// TIA Portal V16 export
// export: Created 2020-03-06T18:52:04.504784Z, ExportSetting WithDefaults, DisplayName Totally Integrated Automation Portal, DisplayVersion V16, DisplayName TIA Portal Version Control Interface, DisplayVersion V16, DisplayName TIA Portal Openness, DisplayVersion V16, DisplayName TIA Portal Teamcenter Gateway, DisplayVersion V16, DisplayName SINAMICS Startdrive Advanced, DisplayVersion V16 Update 1, DisplayName SINAMICS Startdrive G130, G150, S120, S150, SINAMICS MV, S210, DisplayVersion V16 Update 1, DisplayName SINAMICS Startdrive G110M, G120, G120C, G120D, G120P, DisplayVersion V16 Update 1, DisplayName STEP 7 Professional, DisplayVersion V16, DisplayName STEP 7 Safety, DisplayVersion V16, DisplayName WinCC Professional, DisplayVersion V16
FUNCTION_BLOCK "3oo6 AI"   // FB37, LAD
{ S7_Optimized_Access := 'TRUE' }
VERSION : 0.1
// stored: AutoNumber true, IsIECCheckEnabled false, IsRetainMemResEnabled false, MemoryReserve 100, SetENOAutomatically false, UDAEnableTagReadback false
   VAR_INPUT
      V1GA : Bool;   // Value 1
      V2GA : Bool;   // Value 2
      V3GA : Bool;   // Value 3
      V4GA : Bool;
      V5GA : Bool;
      V6GA : Bool;
      "AL.HH3oo6" : Bool;
      "AL.H3oo6" : Bool;
      "AL.L3oo6" : Bool;
      "AL.LL3oo6" : Bool;
      PM : Int;   // Permissive Mode - "0=No P""1=Bool P" "2=Real P"
      HPB : Bool := TRUE;   // High Permissive BOOL
      LPB : Bool := TRUE;   // Low Permissive BOOL
      HPR : Real;   // High Permissive REAL
      LPR : Real;   // Low Permissive REAL
   END_VAR
   VAR_OUTPUT
      V1GA_1 : Bool;   // Value 1
      V2GA_1 : Bool;   // Value 2
      V3GA_1 : Bool;   // Value 3
      V4GA_1 : Bool;
      V5GA_1 : Bool;
      V6GA_1 : Bool;
      "AL.HH_3oo6" : Bool;
      "AL.H_3oo6" : Bool;
      "AL.L_3oo6" : Bool;
      "AL.LL_3oo6" : Bool;
   END_VAR
   VAR DB_SPECIFIC
      Config : Struct   // Configurations
         Limits : Struct
            HH : Real := 100.0;   // High High Limit
            H : Real := 90.0;   // High Limit
            L : Real := 10.0;   // Low Limit
            LL : Real := 5.0;   // Low Low Limit
         END_STRUCT;
         H : Real := 1.0;   // Hysteresis
      END_STRUCT;
      Alarms : Struct
         HH : Bool;   // High High
         H : Bool;   // High
         L : Bool;   // Low
         LL : Bool;   // Low Low
         V1GA : Bool;   // Value 1 General Alarm
         V2GA : Bool;   // Value 2 General Alarm
         V3GA : Bool;   // Value 3 General Alarm
         V4GA : Bool;
         V5GA : Bool;
         V6GA : Bool;
      END_STRUCT;
   END_VAR
   VAR
      V1HHA { ExternalAccessible := 'False'; ExternalVisible := 'False'; ExternalWritable := 'False'} : "HLR";   // Value 1 High High Alarm
      V1HA { ExternalAccessible := 'False'; ExternalVisible := 'False'; ExternalWritable := 'False'} : "HLR";   // Value 1 High Alarm
      V1LA { ExternalAccessible := 'False'; ExternalVisible := 'False'; ExternalWritable := 'False'} : "LLR";   // Value 1 Low Alarm
      V1LLA { ExternalAccessible := 'False'; ExternalVisible := 'False'; ExternalWritable := 'False'} : "LLR";   // Value 1 Low Low Alarm
      V2HHA { ExternalAccessible := 'False'; ExternalVisible := 'False'; ExternalWritable := 'False'} : "HLR";   // Value 2 High High Alarm
      V2HA { ExternalAccessible := 'False'; ExternalVisible := 'False'; ExternalWritable := 'False'} : "HLR";   // Value 2 High Alarm
      V2LA { ExternalAccessible := 'False'; ExternalVisible := 'False'; ExternalWritable := 'False'} : "LLR";   // Value 2 Low Alarm
      V2LLA { ExternalAccessible := 'False'; ExternalVisible := 'False'; ExternalWritable := 'False'} : "LLR";   // Value 2 Low Low Alarm
      V3HHA { ExternalAccessible := 'False'; ExternalVisible := 'False'; ExternalWritable := 'False'} : "HLR";   // Value 3 High High Alarm
      V3HA { ExternalAccessible := 'False'; ExternalVisible := 'False'; ExternalWritable := 'False'} : "HLR";   // Value 3 High Alarm
      V3LA { ExternalAccessible := 'False'; ExternalVisible := 'False'; ExternalWritable := 'False'} : "LLR";   // Value 3 Low Alarm
      V3LLA { ExternalAccessible := 'False'; ExternalVisible := 'False'; ExternalWritable := 'False'} : "LLR";   // Value 3 Low Low Alarm
   END_VAR
   VAR DB_SPECIFIC
      "HMI.FVR" : Real := 100.0;
      "FVR.HH" : DInt;
      "FVR.H" : DInt;
      "FVR.L" : DInt;
      "FVR.LL" : DInt;
      "FVR.HPR" : DInt;
      "FVR.LPR" : DInt;
      "FVR.CONFIG.H" : DInt;
   END_VAR
   VAR
      V4HHA { ExternalAccessible := 'False'; ExternalVisible := 'False'; ExternalWritable := 'False'} : "HLR";
      V4HA { ExternalAccessible := 'False'; ExternalVisible := 'False'; ExternalWritable := 'False'} : "HLR";
      V4LA { ExternalAccessible := 'False'; ExternalVisible := 'False'; ExternalWritable := 'False'} : "LLR";
      V4LLA { ExternalAccessible := 'False'; ExternalVisible := 'False'; ExternalWritable := 'False'} : "LLR";
      V6LLA { ExternalAccessible := 'False'; ExternalVisible := 'False'; ExternalWritable := 'False'} : "LLR";
      V6LA { ExternalAccessible := 'False'; ExternalVisible := 'False'; ExternalWritable := 'False'} : "LLR";
      V6HA { ExternalAccessible := 'False'; ExternalVisible := 'False'; ExternalWritable := 'False'} : "HLR";
      V6HHA { ExternalAccessible := 'False'; ExternalVisible := 'False'; ExternalWritable := 'False'} : "HLR";
      V5LLA { ExternalAccessible := 'False'; ExternalVisible := 'False'; ExternalWritable := 'False'} : "LLR";
      V5LA { ExternalAccessible := 'False'; ExternalVisible := 'False'; ExternalWritable := 'False'} : "LLR";
      V5HA { ExternalAccessible := 'False'; ExternalVisible := 'False'; ExternalWritable := 'False'} : "HLR";
      V5HHA { ExternalAccessible := 'False'; ExternalVisible := 'False'; ExternalWritable := 'False'} : "HLR";
   END_VAR
   VAR_TEMP
      HH123 : Bool;
      HH124 : Bool;
      HH134 : Bool;
      HH234 : Bool;
      HH125 : Bool;
      HH135 : Bool;
      HH235 : Bool;
      HH145 : Bool;
      HH245 : Bool;
      HH345 : Bool;
      HH126 : Bool;
      HH136 : Bool;
      HH236 : Bool;
      HH146 : Bool;
      HH246 : Bool;
      HH346 : Bool;
      HH156 : Bool;
      HH256 : Bool;
      HH356 : Bool;
      HH456 : Bool;
      H123 : Bool;
      H124 : Bool;
      H134 : Bool;
      H234 : Bool;
      H125 : Bool;
      H135 : Bool;
      H235 : Bool;
      H145 : Bool;
      H245 : Bool;
      H345 : Bool;
      H126 : Bool;
      H136 : Bool;
      H236 : Bool;
      H146 : Bool;
      H246 : Bool;
      H346 : Bool;
      H156 : Bool;
      H256 : Bool;
      H356 : Bool;
      H456 : Bool;
      L123 : Bool;
      L124 : Bool;
      L134 : Bool;
      L234 : Bool;
      L125 : Bool;
      L135 : Bool;
      L235 : Bool;
      L145 : Bool;
      L245 : Bool;
      L345 : Bool;
      L126 : Bool;
      L136 : Bool;
      L236 : Bool;
      L146 : Bool;
      L246 : Bool;
      L346 : Bool;
      L156 : Bool;
      L256 : Bool;
      L356 : Bool;
      L456 : Bool;
      LL123 : Bool;
      LL124 : Bool;
      LL134 : Bool;
      LL234 : Bool;
      LL125 : Bool;
      LL135 : Bool;
      LL235 : Bool;
      LL145 : Bool;
      LL245 : Bool;
      LL345 : Bool;
      LL126 : Bool;
      LL136 : Bool;
      LL236 : Bool;
      LL146 : Bool;
      LL246 : Bool;
      LL346 : Bool;
      LL156 : Bool;
      LL256 : Bool;
      LL356 : Bool;
      LL456 : Bool;
      "MATH.HH" : Real;
      "MATH.H" : Real;
      "MATH.LL" : Real;
      "MATH.L" : Real;
      "MATH.HR" : Real;
      "MATH.LR" : Real;
      "MATH.CONFIG.H" : Real;
   END_VAR
BEGIN

REGION Network 1
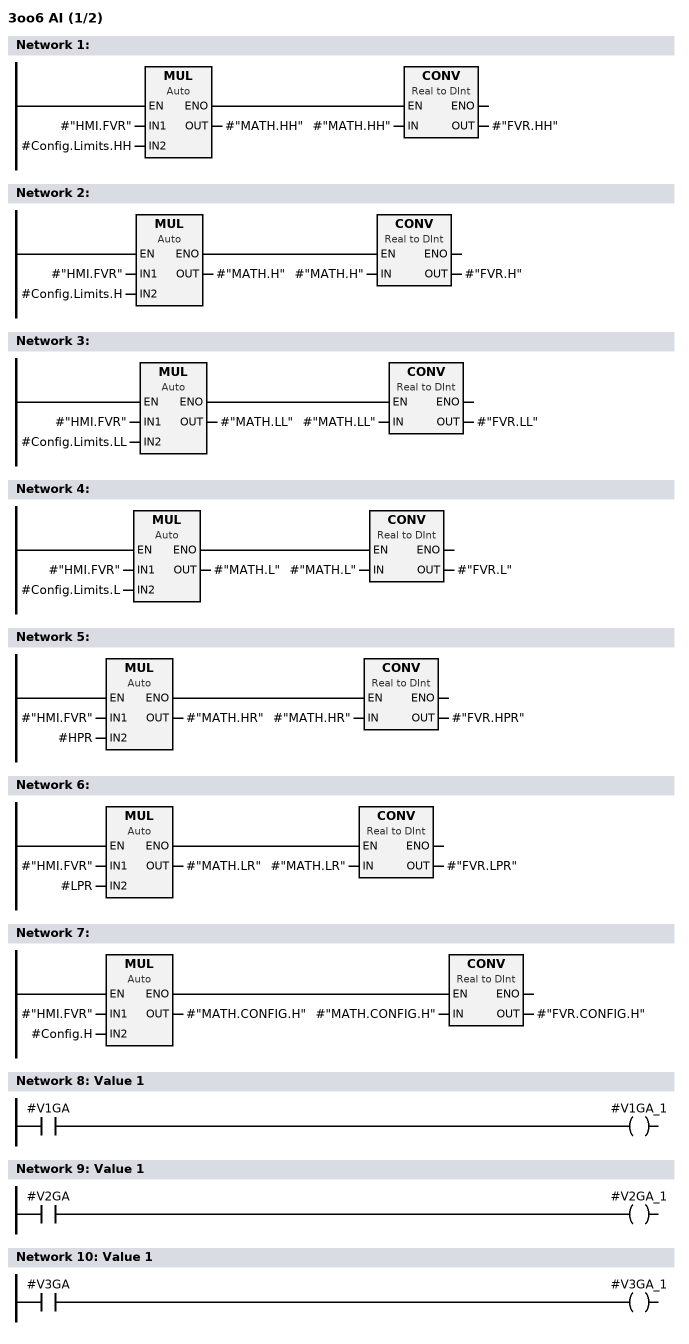
   RUNG wire#powerrail
      Mul(in1 := #"HMI.FVR", in2 := #Config.Limits.HH, out => #"MATH.HH")
      { S7_Templates := "[SrcType := Real, DestType := DInt]" } Convert(in := #"MATH.HH", out => #"FVR.HH")
   END_RUNG
   // the same network as SCL:
   #"MATH.HH" := #"HMI.FVR" * #Config.Limits.HH;
   #"FVR.HH" := REAL_TO_DINT(#"MATH.HH");
END_REGION

REGION Network 2
   RUNG wire#powerrail
      Mul(in1 := #"HMI.FVR", in2 := #Config.Limits.H, out => #"MATH.H")
      { S7_Templates := "[SrcType := Real, DestType := DInt]" } Convert(in := #"MATH.H", out => #"FVR.H")
   END_RUNG
   // the same network as SCL:
   #"MATH.H" := #"HMI.FVR" * #Config.Limits.H;
   #"FVR.H" := REAL_TO_DINT(#"MATH.H");
END_REGION

REGION Network 3
   RUNG wire#powerrail
      Mul(in1 := #"HMI.FVR", in2 := #Config.Limits.LL, out => #"MATH.LL")
      { S7_Templates := "[SrcType := Real, DestType := DInt]" } Convert(in := #"MATH.LL", out => #"FVR.LL")
   END_RUNG
   // the same network as SCL:
   #"MATH.LL" := #"HMI.FVR" * #Config.Limits.LL;
   #"FVR.LL" := REAL_TO_DINT(#"MATH.LL");
END_REGION

REGION Network 4
   RUNG wire#powerrail
      Mul(in1 := #"HMI.FVR", in2 := #Config.Limits.L, out => #"MATH.L")
      { S7_Templates := "[SrcType := Real, DestType := DInt]" } Convert(in := #"MATH.L", out => #"FVR.L")
   END_RUNG
   // the same network as SCL:
   #"MATH.L" := #"HMI.FVR" * #Config.Limits.L;
   #"FVR.L" := REAL_TO_DINT(#"MATH.L");
END_REGION

REGION Network 5
   RUNG wire#powerrail
      Mul(in1 := #"HMI.FVR", in2 := #HPR, out => #"MATH.HR")
      { S7_Templates := "[SrcType := Real, DestType := DInt]" } Convert(in := #"MATH.HR", out => #"FVR.HPR")
   END_RUNG
   // the same network as SCL:
   #"MATH.HR" := #"HMI.FVR" * #HPR;
   #"FVR.HPR" := REAL_TO_DINT(#"MATH.HR");
END_REGION

REGION Network 6
   RUNG wire#powerrail
      Mul(in1 := #"HMI.FVR", in2 := #LPR, out => #"MATH.LR")
      { S7_Templates := "[SrcType := Real, DestType := DInt]" } Convert(in := #"MATH.LR", out => #"FVR.LPR")
   END_RUNG
   // the same network as SCL:
   #"MATH.LR" := #"HMI.FVR" * #LPR;
   #"FVR.LPR" := REAL_TO_DINT(#"MATH.LR");
END_REGION

REGION Network 7
   RUNG wire#powerrail
      Mul(in1 := #"HMI.FVR", in2 := #Config.H, out => #"MATH.CONFIG.H")
      { S7_Templates := "[SrcType := Real, DestType := DInt]" } Convert(in := #"MATH.CONFIG.H", out => #"FVR.CONFIG.H")
   END_RUNG
   // the same network as SCL:
   #"MATH.CONFIG.H" := #"HMI.FVR" * #Config.H;
   #"FVR.CONFIG.H" := REAL_TO_DINT(#"MATH.CONFIG.H");
END_REGION

REGION Network 8: Value 1
   RUNG wire#powerrail
      Contact( #V1GA )
      Coil( #V1GA_1 )
   END_RUNG
   // the same network as SCL:
   #V1GA_1 := #V1GA;
END_REGION

REGION Network 9: Value 1
   RUNG wire#powerrail
      Contact( #V2GA )
      Coil( #V2GA_1 )
   END_RUNG
   // the same network as SCL:
   #V2GA_1 := #V2GA;
END_REGION

REGION Network 10: Value 1
   RUNG wire#powerrail
      Contact( #V3GA )
      Coil( #V3GA_1 )
   END_RUNG
   // the same network as SCL:
   #V3GA_1 := #V3GA;
END_REGION

REGION Network 11: Value 1
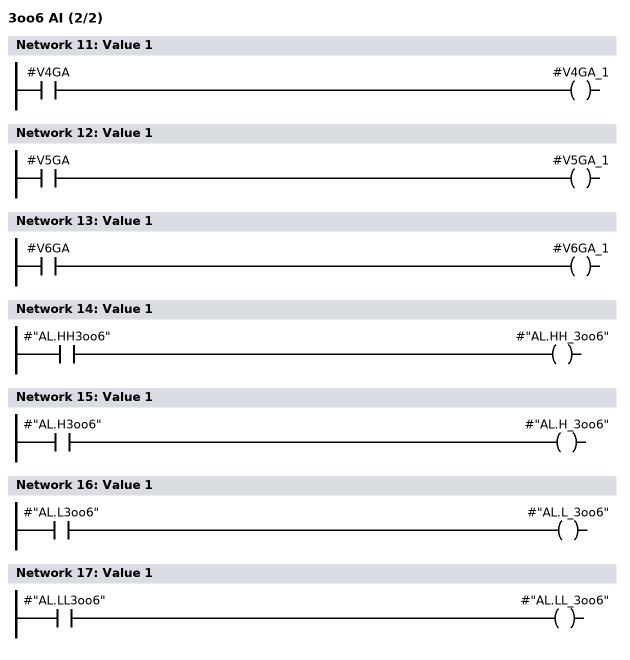
   RUNG wire#powerrail
      Contact( #V4GA )
      Coil( #V4GA_1 )
   END_RUNG
   // the same network as SCL:
   #V4GA_1 := #V4GA;
END_REGION

REGION Network 12: Value 1
   RUNG wire#powerrail
      Contact( #V5GA )
      Coil( #V5GA_1 )
   END_RUNG
   // the same network as SCL:
   #V5GA_1 := #V5GA;
END_REGION

REGION Network 13: Value 1
   RUNG wire#powerrail
      Contact( #V6GA )
      Coil( #V6GA_1 )
   END_RUNG
   // the same network as SCL:
   #V6GA_1 := #V6GA;
END_REGION

REGION Network 14: Value 1
   RUNG wire#powerrail
      Contact( #"AL.HH3oo6" )
      Coil( #"AL.HH_3oo6" )
   END_RUNG
   // the same network as SCL:
   #"AL.HH_3oo6" := #"AL.HH3oo6";
END_REGION

REGION Network 15: Value 1
   RUNG wire#powerrail
      Contact( #"AL.H3oo6" )
      Coil( #"AL.H_3oo6" )
   END_RUNG
   // the same network as SCL:
   #"AL.H_3oo6" := #"AL.H3oo6";
END_REGION

REGION Network 16: Value 1
   RUNG wire#powerrail
      Contact( #"AL.L3oo6" )
      Coil( #"AL.L_3oo6" )
   END_RUNG
   // the same network as SCL:
   #"AL.L_3oo6" := #"AL.L3oo6";
END_REGION

REGION Network 17: Value 1
   RUNG wire#powerrail
      Contact( #"AL.LL3oo6" )
      Coil( #"AL.LL_3oo6" )
   END_RUNG
   // the same network as SCL:
   #"AL.LL_3oo6" := #"AL.LL3oo6";
END_REGION
END_FUNCTION_BLOCK
